INTERFACE I_ParameterPositionGetter EXTENDS I_Base

{attribute 'monitoring' := 'call'}
PROPERTY Position : LREAL
GET
END_GET
END_PROPERTY

END_INTERFACE

(* stored: Version 1.1.0.1
   Itf I_ParameterPositionGetter: Id {10703703-a0d9-4fc8-b31a-8c1d3da1f916}
   Property Position: Id {6ebfa236-c9a7-4610-b5ce-1616d65ee0bc}
   Get Get: Id {9f58f3f7-e161-4378-b5be-18e5146e0b0e} *)
